// SIMATIC S7-200 project (STEP 7-Micro/WIN), CPU 224 REL 02.01

SYMBOL_TABLE USER1
start            I0.0
stopp            I0.1
tlb1             I0.2
tlb2             I0.3
reset            I0.4
motor            Q0.0
mv1              Q0.1
mv2              Q0.2
END_SYMBOL_TABLE

ORGANIZATION_BLOCK MAIN:OB1
TITLE=PROGRAM COMMENTS
BEGIN
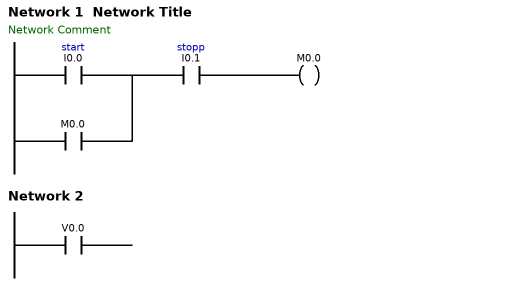
Network 1 // Network Title
// Network Comment
// (network saved uncompiled; LAD cells follow)
// row 0: c0 -| |- start:I0.0 v  c1 -| |- stopp:I0.1  c2 -( ) M0.0
// row 1: c0 -| |- M0.0 ^
Network 2
// (network saved uncompiled; LAD cells follow)
// row 0: c0 -| |- V0.0
END_ORGANIZATION_BLOCK
